{attribute 'Tc2GvlVarNames'}
{attribute 'strict'}
TYPE e_ProgrammiMovimentoJ :
(
	
	J_PosDiRiposo						:= 0,
	J_PosFuoriIngombro					:= 6,

	J_PosPrelievoFalda					:= 10,
	J_PosDepositoFalda					:= 11,
	
	J_PosPrelievoLastra					:= 12,
	J_PosDepositoLastra					:= 13,
	J_PosStartApproccioPrelLastra		:= 14,
	J_PosSfogliatura					:= 15,
	
	J_PosStartDepLastra					:= 16,
	
	J_PosPostScarico					:= 17,

	J_PosFuoriIngombroPosAttuale		:= 18

	
);
END_TYPE

(* stored: Version 1.1.0.1, ProductVersion 3.1.4024.11
   EnumerationTextList e_ProgrammiMovimentoJ: Id {f9c552f1-0b98-423c-b466-ef2960be12d4} *)
